FUNCTION_BLOCK EL3022
VAR
	_io : EL3xx2_Data;
	{attribute addProperty Name "WcState"}
	_wcState : WcStateInputToggle;
	{attribute addProperty Name "Info data"}
	_infoData : InfoDataAds;
END_VAR

PROPERTY IO : REFERENCE TO EL3xx2_Data
GET
IO REF= _io;
END_GET
END_PROPERTY

PROPERTY WcState : REFERENCE TO WcStateInputToggle
GET
WcState REF= _wcState;
END_GET
END_PROPERTY

END_FUNCTION_BLOCK

(* stored: Version 1.1.0.1, ProductVersion 3.1.4024.9
   POU EL3022: Id {fd194cae-face-0f99-23ac-a88f572ee16d}, SpecialFunc None
   Property IO: Id {03fa7585-9304-0b2d-1123-4e0df9c59df3}
   Get Get: Id {8487a004-147c-0dea-2081-b61298dd0e2f}
   Property WcState: Id {96088c07-92c7-00f8-2883-0bad4dc3699a}
   Get Get: Id {284bd9b3-16fa-00eb-08ce-6e4ca159031a} *)
